TYPE "LubrMotor_Alr"
VERSION : 0.1
// Block: LubrMotor_Alr
   STRUCT
      RotationFeedback : Bool;
      LowLevelLubrication : Bool;
      MotorAlr : MotorAlr;
   END_STRUCT;

END_TYPE
